// TIA Portal project "pick and place xyz" (V17)
// Vorlageprojekt für das Buch mit Zielsystem S7-1200

(* hardware
DEVICE "S7-1200-Station_1"  S7-1200 Station
   slot 0: "Baugruppenträger_0"  Rack  V1.0
   slot 1: "PLC_1"  CPU 1211C DC/DC/DC  6ES7 211-1AE40-0XB0  V4.1
*)

// ===== PLC "PLC_1"  CPU 1211C DC/DC/DC =====

VAR_GLOBAL   // PLC tag table "Standard-Variablentabelle"
   "box at place" AT %I0.0 : Bool;
   "part at place" AT %I0.1 : Bool;
   "detected" AT %I0.2 : Bool;
   "c limit" AT %I0.3 : Bool;
   "start" AT %I0.4 : Bool;
   "reset" AT %I0.5 : Bool;
   "stop" AT %I0.6 : Bool;
   "e stop" AT %I0.7 : Bool;
   "auto" AT %I1.0 : Bool;
   "FACTORY io run" AT %I1.1 : Bool;
   "x" AT %ID30 : Real;
   "y" AT %ID34 : Real;
   "z" AT %ID38 : Real;
   "box conv" AT %Q0.0 : Bool;
   "part conv" AT %Q0.1 : Bool;
   "exit conv" AT %Q0.2 : Bool;
   "c+" AT %Q0.3 : Bool;
   "grab" AT %Q0.4 : Bool;
   "exit green" AT %Q0.5 : Bool;
   "exit yellow" AT %Q0.6 : Bool;
   "exit red" AT %Q0.7 : Bool;
   "start light" AT %Q1.0 : Bool;
   "reset light" AT %Q1.1 : Bool;
   "stop light" AT %Q1.2 : Bool;
   "sp x" AT %QD30 : Real;
   "sp y" AT %QD34 : Real;
   "sp z" AT %QD38 : Real;
   "count" AT %QD42 : DInt;
   "Tag_1" AT %M0.0 : Bool;
   "Tag_2" AT %M0.1 : Bool;
   "reset count" AT %M0.2 : Bool;
END_VAR

DATA_BLOCK "modes"   // DB2
{ S7_Optimized_Access := 'TRUE' }
VERSION : 0.1
   VAR
      "stop mode" : Bool;
      "start mode" : Bool;
      "auto mode" : Bool;
      "reset mode" : Bool;
      "e stop mode" : Bool;
      "home position" : Bool;
   END_VAR
BEGIN
END_DATA_BLOCK

DATA_BLOCK "steps"   // DB4
{ S7_Optimized_Access := 'TRUE' }
VERSION : 0.1
   VAR
      "next step" : Int := 0;
      "curent step" : Int := 0;
   END_VAR
BEGIN
END_DATA_BLOCK

// folder: System blocks/Program resources

DATA_BLOCK "counter"   // DB1
{ S7_Optimized_Access := 'TRUE' }
AUTHOR : Simatic
FAMILY : IEC
NAME : CNTR
VERSION : 1.0
// stored: InstanceOfName IEC_COUNTER
"IEC_COUNTER"
BEGIN
END_DATA_BLOCK

// folder: (top level)

FUNCTION "1 operation modes" : Void   // FC1, LAD
{ S7_Optimized_Access := 'TRUE' }
VERSION : 0.1
BEGIN

REGION Network 1: start mode
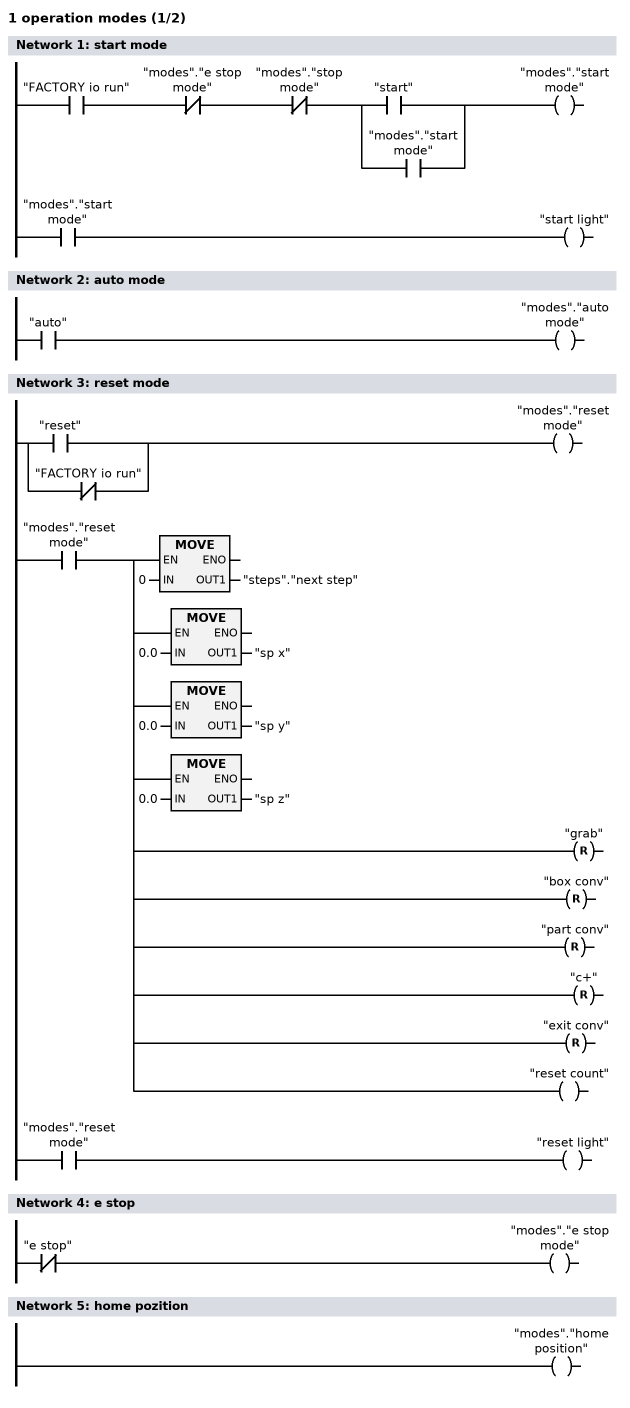
   RUNG wire#powerrail
      Contact( "FACTORY io run" )
      I_Contact( "modes"."e stop mode" )
      I_Contact( "modes"."stop mode" )
      wire#w1
      Contact( "start" )
      wire#w2
      Coil( "modes"."start mode" )
   END_RUNG
   RUNG wire#w1
      Contact( "modes"."start mode" )
   END_RUNG wire#w2
   RUNG wire#powerrail
      Contact( "modes"."start mode" )
      Coil( "start light" )
   END_RUNG
   // the same network as SCL:
   "modes"."start mode" := "FACTORY io run" AND NOT "modes"."e stop mode" AND NOT "modes"."stop mode" AND ("start" OR "modes"."start mode");
   "start light" := "modes"."start mode";
END_REGION

REGION Network 2: auto mode
   RUNG wire#powerrail
      Contact( "auto" )
      Coil( "modes"."auto mode" )
   END_RUNG
   // the same network as SCL:
   "modes"."auto mode" := "auto";
END_REGION

REGION Network 3: reset mode
   RUNG wire#powerrail
      Contact( "reset" )
      wire#w1
      Coil( "modes"."reset mode" )
   END_RUNG
   RUNG wire#powerrail
      I_Contact( "FACTORY io run" )
   END_RUNG wire#w1
   RUNG wire#powerrail
      Contact( "modes"."reset mode" )
      wire#w2
      Move(in := 0, out1 => "steps"."next step")
   END_RUNG
   RUNG wire#w2
      Move(in := 0.0, out1 => "sp x")
   END_RUNG
   RUNG wire#w2
      Move(in := 0.0, out1 => "sp y")
   END_RUNG
   RUNG wire#w2
      Move(in := 0.0, out1 => "sp z")
   END_RUNG
   RUNG wire#w2
      R_Coil( "grab" )
   END_RUNG
   RUNG wire#w2
      R_Coil( "box conv" )
   END_RUNG
   RUNG wire#w2
      R_Coil( "part conv" )
   END_RUNG
   RUNG wire#w2
      R_Coil( "c+" )
   END_RUNG
   RUNG wire#w2
      R_Coil( "exit conv" )
   END_RUNG
   RUNG wire#w2
      Coil( "reset count" )
   END_RUNG
   RUNG wire#powerrail
      Contact( "modes"."reset mode" )
      Coil( "reset light" )
   END_RUNG
   // the same network as SCL:
   "modes"."reset mode" := "reset" OR NOT "FACTORY io run";
   IF "modes"."reset mode" THEN
       "steps"."next step" := 0;
       "sp x" := 0.0;
       "sp y" := 0.0;
       "sp z" := 0.0;
       "grab" := FALSE;
       "box conv" := FALSE;
       "part conv" := FALSE;
       "c+" := FALSE;
       "exit conv" := FALSE;
   END_IF;
   "reset count" := "modes"."reset mode";
   "reset light" := "modes"."reset mode";
END_REGION

REGION Network 4: e stop
   RUNG wire#powerrail
      I_Contact( "e stop" )
      Coil( "modes"."e stop mode" )
   END_RUNG
   // the same network as SCL:
   "modes"."e stop mode" := NOT "e stop";
END_REGION

REGION Network 5: home pozition
   RUNG wire#powerrail
      Coil( "modes"."home position" )
   END_RUNG
   // the same network as SCL:
   "modes"."home position" := TRUE;
END_REGION

REGION Network 6
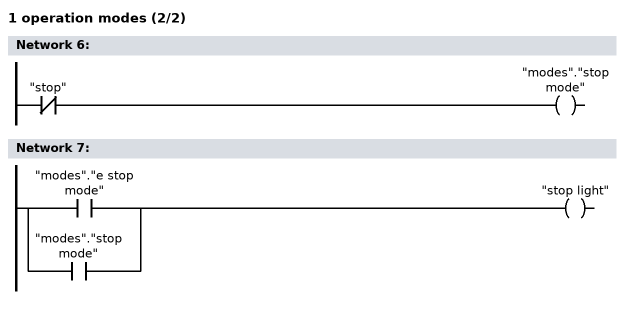
   RUNG wire#powerrail
      I_Contact( "stop" )
      Coil( "modes"."stop mode" )
   END_RUNG
   // the same network as SCL:
   "modes"."stop mode" := NOT "stop";
END_REGION

REGION Network 7
   RUNG wire#powerrail
      Contact( "modes"."e stop mode" )
      wire#w1
      Coil( "stop light" )
   END_RUNG
   RUNG wire#powerrail
      Contact( "modes"."stop mode" )
   END_RUNG wire#w1
   // the same network as SCL:
   "stop light" := "modes"."e stop mode" OR "modes"."stop mode";
END_REGION
END_FUNCTION

FUNCTION "2 step definition" : Void   // FC2, LAD
{ S7_Optimized_Access := 'TRUE' }
VERSION : 0.1
BEGIN

REGION Network 1
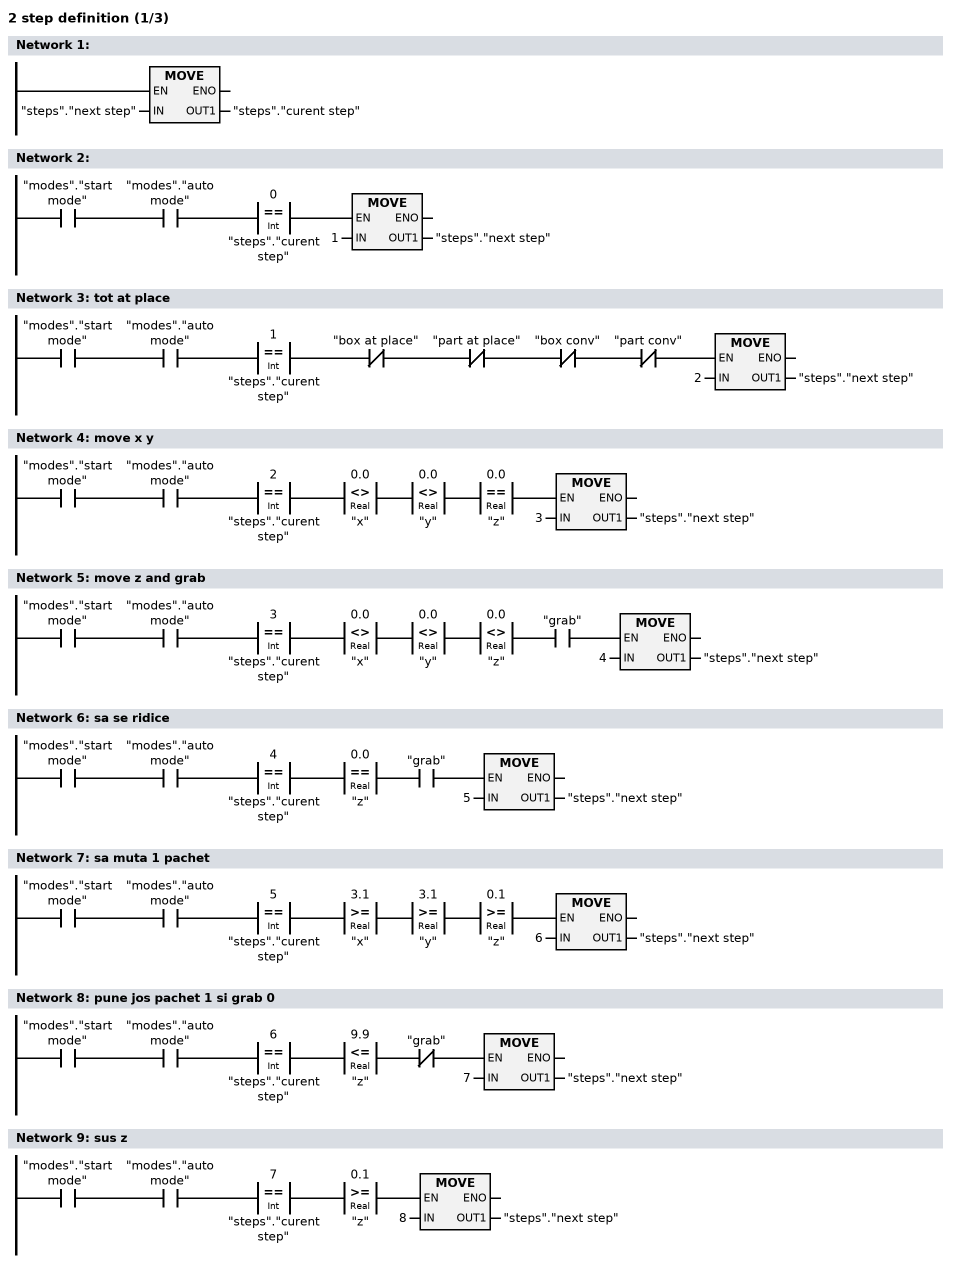
   RUNG wire#powerrail
      Move(in := "steps"."next step", out1 => "steps"."curent step")
   END_RUNG
   // the same network as SCL:
   "steps"."curent step" := "steps"."next step";
END_REGION

REGION Network 2
   RUNG wire#powerrail
      Contact( "modes"."start mode" )
      Contact( "modes"."auto mode" )
      { S7_Templates := "SrcType := Int" } EQ_Contact(in1 := 0, in2 := "steps"."curent step")
      Move(in := 1, out1 => "steps"."next step")
   END_RUNG
   // the same network as SCL:
   IF "modes"."start mode" AND "modes"."auto mode" AND (0 = "steps"."curent step") THEN
       "steps"."next step" := 1;
   END_IF;
END_REGION

REGION Network 3: tot at place
   RUNG wire#powerrail
      Contact( "modes"."start mode" )
      Contact( "modes"."auto mode" )
      { S7_Templates := "SrcType := Int" } EQ_Contact(in1 := 1, in2 := "steps"."curent step")
      I_Contact( "box at place" )
      I_Contact( "part at place" )
      I_Contact( "box conv" )
      I_Contact( "part conv" )
      Move(in := 2, out1 => "steps"."next step")
   END_RUNG
   // the same network as SCL:
   IF "modes"."start mode" AND "modes"."auto mode" AND (1 = "steps"."curent step") AND NOT "box at place" AND NOT "part at place" AND NOT "box conv" AND NOT "part conv" THEN
       "steps"."next step" := 2;
   END_IF;
END_REGION

REGION Network 4: move x y
   RUNG wire#powerrail
      Contact( "modes"."start mode" )
      Contact( "modes"."auto mode" )
      { S7_Templates := "SrcType := Int" } EQ_Contact(in1 := 2, in2 := "steps"."curent step")
      { S7_Templates := "SrcType := Real" } NE_Contact(in1 := 0.0, in2 := "x")
      { S7_Templates := "SrcType := Real" } NE_Contact(in1 := 0.0, in2 := "y")
      { S7_Templates := "SrcType := Real" } EQ_Contact(in1 := 0.0, in2 := "z")
      Move(in := 3, out1 => "steps"."next step")
   END_RUNG
   // the same network as SCL:
   IF "modes"."start mode" AND "modes"."auto mode" AND (2 = "steps"."curent step") AND (0.0 <> "x") AND (0.0 <> "y") AND (0.0 = "z") THEN
       "steps"."next step" := 3;
   END_IF;
END_REGION

REGION Network 5: move z and grab
   RUNG wire#powerrail
      Contact( "modes"."start mode" )
      Contact( "modes"."auto mode" )
      { S7_Templates := "SrcType := Int" } EQ_Contact(in1 := 3, in2 := "steps"."curent step")
      { S7_Templates := "SrcType := Real" } NE_Contact(in1 := 0.0, in2 := "x")
      { S7_Templates := "SrcType := Real" } NE_Contact(in1 := 0.0, in2 := "y")
      { S7_Templates := "SrcType := Real" } NE_Contact(in1 := 0.0, in2 := "z")
      Contact( "grab" )
      Move(in := 4, out1 => "steps"."next step")
   END_RUNG
   // the same network as SCL:
   IF "modes"."start mode" AND "modes"."auto mode" AND (3 = "steps"."curent step") AND (0.0 <> "x") AND (0.0 <> "y") AND (0.0 <> "z") AND "grab" THEN
       "steps"."next step" := 4;
   END_IF;
END_REGION

REGION Network 6: sa se ridice
   RUNG wire#powerrail
      Contact( "modes"."start mode" )
      Contact( "modes"."auto mode" )
      { S7_Templates := "SrcType := Int" } EQ_Contact(in1 := 4, in2 := "steps"."curent step")
      { S7_Templates := "SrcType := Real" } EQ_Contact(in1 := 0.0, in2 := "z")
      Contact( "grab" )
      Move(in := 5, out1 => "steps"."next step")
   END_RUNG
   // the same network as SCL:
   IF "modes"."start mode" AND "modes"."auto mode" AND (4 = "steps"."curent step") AND (0.0 = "z") AND "grab" THEN
       "steps"."next step" := 5;
   END_IF;
END_REGION

REGION Network 7: sa muta 1 pachet
   RUNG wire#powerrail
      Contact( "modes"."start mode" )
      Contact( "modes"."auto mode" )
      { S7_Templates := "SrcType := Int" } EQ_Contact(in1 := 5, in2 := "steps"."curent step")
      { S7_Templates := "SrcType := Real" } GE_Contact(in1 := 3.1, in2 := "x")
      { S7_Templates := "SrcType := Real" } GE_Contact(in1 := 3.1, in2 := "y")
      { S7_Templates := "SrcType := Real" } GE_Contact(in1 := 0.1, in2 := "z")
      Move(in := 6, out1 => "steps"."next step")
   END_RUNG
   // the same network as SCL:
   IF "modes"."start mode" AND "modes"."auto mode" AND (5 = "steps"."curent step") AND (3.1 >= "x") AND (3.1 >= "y") AND (0.1 >= "z") THEN
       "steps"."next step" := 6;
   END_IF;
END_REGION

REGION Network 8: pune jos pachet 1 si grab 0
   RUNG wire#powerrail
      Contact( "modes"."start mode" )
      Contact( "modes"."auto mode" )
      { S7_Templates := "SrcType := Int" } EQ_Contact(in1 := 6, in2 := "steps"."curent step")
      { S7_Templates := "SrcType := Real" } LE_Contact(in1 := 9.9, in2 := "z")
      I_Contact( "grab" )
      Move(in := 7, out1 => "steps"."next step")
   END_RUNG
   // the same network as SCL:
   IF "modes"."start mode" AND "modes"."auto mode" AND (6 = "steps"."curent step") AND (9.9 <= "z") AND NOT "grab" THEN
       "steps"."next step" := 7;
   END_IF;
END_REGION

REGION Network 9: sus z
   RUNG wire#powerrail
      Contact( "modes"."start mode" )
      Contact( "modes"."auto mode" )
      { S7_Templates := "SrcType := Int" } EQ_Contact(in1 := 7, in2 := "steps"."curent step")
      { S7_Templates := "SrcType := Real" } GE_Contact(in1 := 0.1, in2 := "z")
      Move(in := 8, out1 => "steps"."next step")
   END_RUNG
   // the same network as SCL:
   IF "modes"."start mode" AND "modes"."auto mode" AND (7 = "steps"."curent step") AND (0.1 >= "z") THEN
       "steps"."next step" := 8;
   END_IF;
END_REGION

REGION Network 10: xyz at place
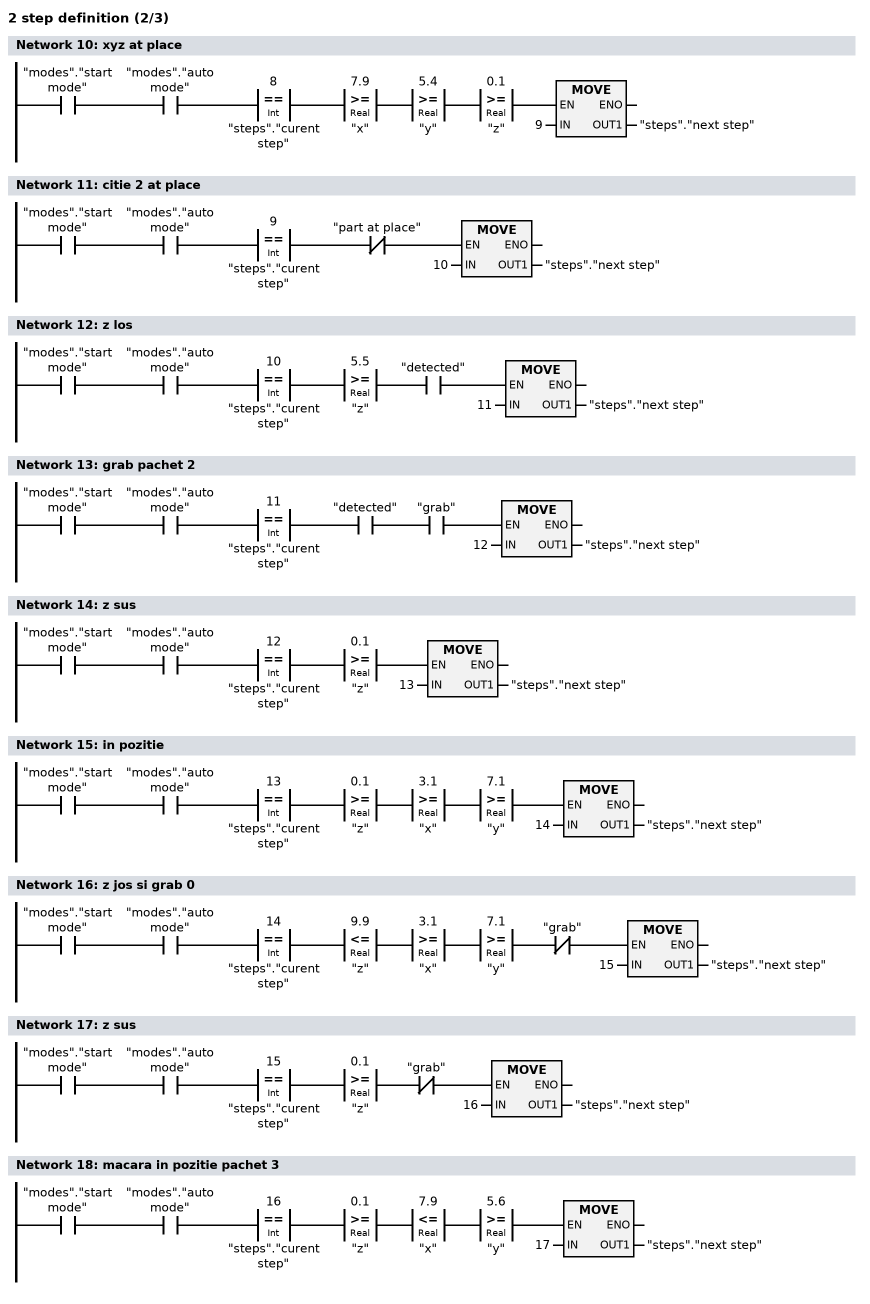
   RUNG wire#powerrail
      Contact( "modes"."start mode" )
      Contact( "modes"."auto mode" )
      { S7_Templates := "SrcType := Int" } EQ_Contact(in1 := 8, in2 := "steps"."curent step")
      { S7_Templates := "SrcType := Real" } GE_Contact(in1 := 7.9, in2 := "x")
      { S7_Templates := "SrcType := Real" } GE_Contact(in1 := 5.4, in2 := "y")
      { S7_Templates := "SrcType := Real" } GE_Contact(in1 := 0.1, in2 := "z")
      Move(in := 9, out1 => "steps"."next step")
   END_RUNG
   // the same network as SCL:
   IF "modes"."start mode" AND "modes"."auto mode" AND (8 = "steps"."curent step") AND (7.9 >= "x") AND (5.4 >= "y") AND (0.1 >= "z") THEN
       "steps"."next step" := 9;
   END_IF;
END_REGION

REGION Network 11: citie 2 at place
   RUNG wire#powerrail
      Contact( "modes"."start mode" )
      Contact( "modes"."auto mode" )
      { S7_Templates := "SrcType := Int" } EQ_Contact(in1 := 9, in2 := "steps"."curent step")
      I_Contact( "part at place" )
      Move(in := 10, out1 => "steps"."next step")
   END_RUNG
   // the same network as SCL:
   IF "modes"."start mode" AND "modes"."auto mode" AND (9 = "steps"."curent step") AND NOT "part at place" THEN
       "steps"."next step" := 10;
   END_IF;
END_REGION

REGION Network 12: z los
   RUNG wire#powerrail
      Contact( "modes"."start mode" )
      Contact( "modes"."auto mode" )
      { S7_Templates := "SrcType := Int" } EQ_Contact(in1 := 10, in2 := "steps"."curent step")
      { S7_Templates := "SrcType := Real" } GE_Contact(in1 := 5.5, in2 := "z")
      Contact( "detected" )
      Move(in := 11, out1 => "steps"."next step")
   END_RUNG
   // the same network as SCL:
   IF "modes"."start mode" AND "modes"."auto mode" AND (10 = "steps"."curent step") AND (5.5 >= "z") AND "detected" THEN
       "steps"."next step" := 11;
   END_IF;
END_REGION

REGION Network 13: grab pachet 2
   RUNG wire#powerrail
      Contact( "modes"."start mode" )
      Contact( "modes"."auto mode" )
      { S7_Templates := "SrcType := Int" } EQ_Contact(in1 := 11, in2 := "steps"."curent step")
      Contact( "detected" )
      Contact( "grab" )
      Move(in := 12, out1 => "steps"."next step")
   END_RUNG
   // the same network as SCL:
   IF "modes"."start mode" AND "modes"."auto mode" AND (11 = "steps"."curent step") AND "detected" AND "grab" THEN
       "steps"."next step" := 12;
   END_IF;
END_REGION

REGION Network 14: z sus
   RUNG wire#powerrail
      Contact( "modes"."start mode" )
      Contact( "modes"."auto mode" )
      { S7_Templates := "SrcType := Int" } EQ_Contact(in1 := 12, in2 := "steps"."curent step")
      { S7_Templates := "SrcType := Real" } GE_Contact(in1 := 0.1, in2 := "z")
      Move(in := 13, out1 => "steps"."next step")
   END_RUNG
   // the same network as SCL:
   IF "modes"."start mode" AND "modes"."auto mode" AND (12 = "steps"."curent step") AND (0.1 >= "z") THEN
       "steps"."next step" := 13;
   END_IF;
END_REGION

REGION Network 15: in pozitie
   RUNG wire#powerrail
      Contact( "modes"."start mode" )
      Contact( "modes"."auto mode" )
      { S7_Templates := "SrcType := Int" } EQ_Contact(in1 := 13, in2 := "steps"."curent step")
      { S7_Templates := "SrcType := Real" } GE_Contact(in1 := 0.1, in2 := "z")
      { S7_Templates := "SrcType := Real" } GE_Contact(in1 := 3.1, in2 := "x")
      { S7_Templates := "SrcType := Real" } GE_Contact(in1 := 7.1, in2 := "y")
      Move(in := 14, out1 => "steps"."next step")
   END_RUNG
   // the same network as SCL:
   IF "modes"."start mode" AND "modes"."auto mode" AND (13 = "steps"."curent step") AND (0.1 >= "z") AND (3.1 >= "x") AND (7.1 >= "y") THEN
       "steps"."next step" := 14;
   END_IF;
END_REGION

REGION Network 16: z jos si grab 0
   RUNG wire#powerrail
      Contact( "modes"."start mode" )
      Contact( "modes"."auto mode" )
      { S7_Templates := "SrcType := Int" } EQ_Contact(in1 := 14, in2 := "steps"."curent step")
      { S7_Templates := "SrcType := Real" } LE_Contact(in1 := 9.9, in2 := "z")
      { S7_Templates := "SrcType := Real" } GE_Contact(in1 := 3.1, in2 := "x")
      { S7_Templates := "SrcType := Real" } GE_Contact(in1 := 7.1, in2 := "y")
      I_Contact( "grab" )
      Move(in := 15, out1 => "steps"."next step")
   END_RUNG
   // the same network as SCL:
   IF "modes"."start mode" AND "modes"."auto mode" AND (14 = "steps"."curent step") AND (9.9 <= "z") AND (3.1 >= "x") AND (7.1 >= "y") AND NOT "grab" THEN
       "steps"."next step" := 15;
   END_IF;
END_REGION

REGION Network 17: z sus
   RUNG wire#powerrail
      Contact( "modes"."start mode" )
      Contact( "modes"."auto mode" )
      { S7_Templates := "SrcType := Int" } EQ_Contact(in1 := 15, in2 := "steps"."curent step")
      { S7_Templates := "SrcType := Real" } GE_Contact(in1 := 0.1, in2 := "z")
      I_Contact( "grab" )
      Move(in := 16, out1 => "steps"."next step")
   END_RUNG
   // the same network as SCL:
   IF "modes"."start mode" AND "modes"."auto mode" AND (15 = "steps"."curent step") AND (0.1 >= "z") AND NOT "grab" THEN
       "steps"."next step" := 16;
   END_IF;
END_REGION

REGION Network 18: macara in pozitie pachet 3
   RUNG wire#powerrail
      Contact( "modes"."start mode" )
      Contact( "modes"."auto mode" )
      { S7_Templates := "SrcType := Int" } EQ_Contact(in1 := 16, in2 := "steps"."curent step")
      { S7_Templates := "SrcType := Real" } GE_Contact(in1 := 0.1, in2 := "z")
      { S7_Templates := "SrcType := Real" } LE_Contact(in1 := 7.9, in2 := "x")
      { S7_Templates := "SrcType := Real" } GE_Contact(in1 := 5.6, in2 := "y")
      Move(in := 17, out1 => "steps"."next step")
   END_RUNG
   // the same network as SCL:
   IF "modes"."start mode" AND "modes"."auto mode" AND (16 = "steps"."curent step") AND (0.1 >= "z") AND (7.9 <= "x") AND (5.6 >= "y") THEN
       "steps"."next step" := 17;
   END_IF;
END_REGION

REGION Network 19: part 3 in pozitie
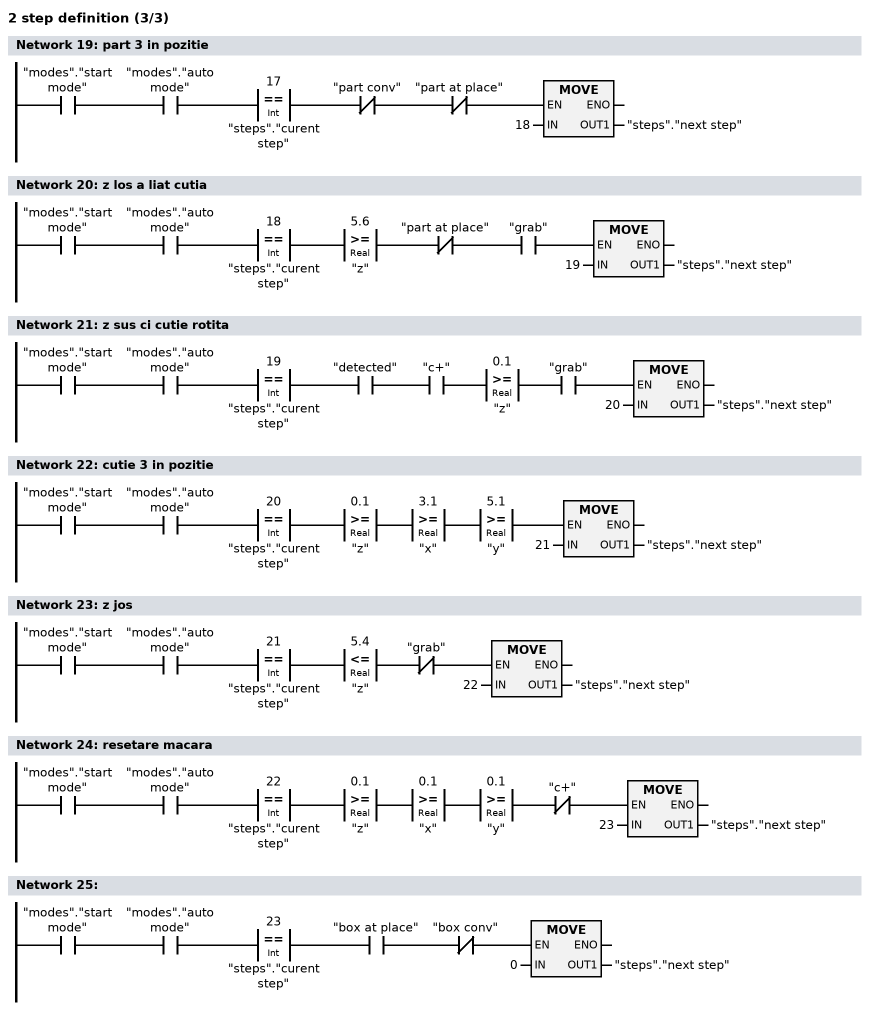
   RUNG wire#powerrail
      Contact( "modes"."start mode" )
      Contact( "modes"."auto mode" )
      { S7_Templates := "SrcType := Int" } EQ_Contact(in1 := 17, in2 := "steps"."curent step")
      I_Contact( "part conv" )
      I_Contact( "part at place" )
      Move(in := 18, out1 => "steps"."next step")
   END_RUNG
   // the same network as SCL:
   IF "modes"."start mode" AND "modes"."auto mode" AND (17 = "steps"."curent step") AND NOT "part conv" AND NOT "part at place" THEN
       "steps"."next step" := 18;
   END_IF;
END_REGION

REGION Network 20: z los a liat cutia
   RUNG wire#powerrail
      Contact( "modes"."start mode" )
      Contact( "modes"."auto mode" )
      { S7_Templates := "SrcType := Int" } EQ_Contact(in1 := 18, in2 := "steps"."curent step")
      { S7_Templates := "SrcType := Real" } GE_Contact(in1 := 5.6, in2 := "z")
      I_Contact( "part at place" )
      Contact( "grab" )
      Move(in := 19, out1 => "steps"."next step")
   END_RUNG
   // the same network as SCL:
   IF "modes"."start mode" AND "modes"."auto mode" AND (18 = "steps"."curent step") AND (5.6 >= "z") AND NOT "part at place" AND "grab" THEN
       "steps"."next step" := 19;
   END_IF;
END_REGION

REGION Network 21: z sus ci cutie rotita
   RUNG wire#powerrail
      Contact( "modes"."start mode" )
      Contact( "modes"."auto mode" )
      { S7_Templates := "SrcType := Int" } EQ_Contact(in1 := 19, in2 := "steps"."curent step")
      Contact( "detected" )
      Contact( "c+" )
      { S7_Templates := "SrcType := Real" } GE_Contact(in1 := 0.1, in2 := "z")
      Contact( "grab" )
      Move(in := 20, out1 => "steps"."next step")
   END_RUNG
   // the same network as SCL:
   IF "modes"."start mode" AND "modes"."auto mode" AND (19 = "steps"."curent step") AND "detected" AND "c+" AND (0.1 >= "z") AND "grab" THEN
       "steps"."next step" := 20;
   END_IF;
END_REGION

REGION Network 22: cutie 3 in pozitie
   RUNG wire#powerrail
      Contact( "modes"."start mode" )
      Contact( "modes"."auto mode" )
      { S7_Templates := "SrcType := Int" } EQ_Contact(in1 := 20, in2 := "steps"."curent step")
      { S7_Templates := "SrcType := Real" } GE_Contact(in1 := 0.1, in2 := "z")
      { S7_Templates := "SrcType := Real" } GE_Contact(in1 := 3.1, in2 := "x")
      { S7_Templates := "SrcType := Real" } GE_Contact(in1 := 5.1, in2 := "y")
      Move(in := 21, out1 => "steps"."next step")
   END_RUNG
   // the same network as SCL:
   IF "modes"."start mode" AND "modes"."auto mode" AND (20 = "steps"."curent step") AND (0.1 >= "z") AND (3.1 >= "x") AND (5.1 >= "y") THEN
       "steps"."next step" := 21;
   END_IF;
END_REGION

REGION Network 23: z jos
   RUNG wire#powerrail
      Contact( "modes"."start mode" )
      Contact( "modes"."auto mode" )
      { S7_Templates := "SrcType := Int" } EQ_Contact(in1 := 21, in2 := "steps"."curent step")
      { S7_Templates := "SrcType := Real" } LE_Contact(in1 := 5.4, in2 := "z")
      I_Contact( "grab" )
      Move(in := 22, out1 => "steps"."next step")
   END_RUNG
   // the same network as SCL:
   IF "modes"."start mode" AND "modes"."auto mode" AND (21 = "steps"."curent step") AND (5.4 <= "z") AND NOT "grab" THEN
       "steps"."next step" := 22;
   END_IF;
END_REGION

REGION Network 24: resetare macara
   RUNG wire#powerrail
      Contact( "modes"."start mode" )
      Contact( "modes"."auto mode" )
      { S7_Templates := "SrcType := Int" } EQ_Contact(in1 := 22, in2 := "steps"."curent step")
      { S7_Templates := "SrcType := Real" } GE_Contact(in1 := 0.1, in2 := "z")
      { S7_Templates := "SrcType := Real" } GE_Contact(in1 := 0.1, in2 := "x")
      { S7_Templates := "SrcType := Real" } GE_Contact(in1 := 0.1, in2 := "y")
      I_Contact( "c+" )
      Move(in := 23, out1 => "steps"."next step")
   END_RUNG
   // the same network as SCL:
   IF "modes"."start mode" AND "modes"."auto mode" AND (22 = "steps"."curent step") AND (0.1 >= "z") AND (0.1 >= "x") AND (0.1 >= "y") AND NOT "c+" THEN
       "steps"."next step" := 23;
   END_IF;
END_REGION

REGION Network 25
   RUNG wire#powerrail
      Contact( "modes"."start mode" )
      Contact( "modes"."auto mode" )
      { S7_Templates := "SrcType := Int" } EQ_Contact(in1 := 23, in2 := "steps"."curent step")
      Contact( "box at place" )
      I_Contact( "box conv" )
      Move(in := 0, out1 => "steps"."next step")
   END_RUNG
   // the same network as SCL:
   IF "modes"."start mode" AND "modes"."auto mode" AND (23 = "steps"."curent step") AND "box at place" AND NOT "box conv" THEN
       "steps"."next step" := 0;
   END_IF;
END_REGION
END_FUNCTION

FUNCTION "3 step execution" : Void   // FC3, LAD
{ S7_Optimized_Access := 'TRUE' }
VERSION : 0.1
   VAR_TEMP   // added for the SCL form of the ladder/FBD networks
      _w1 : Bool;
   END_VAR
BEGIN

REGION Network 1
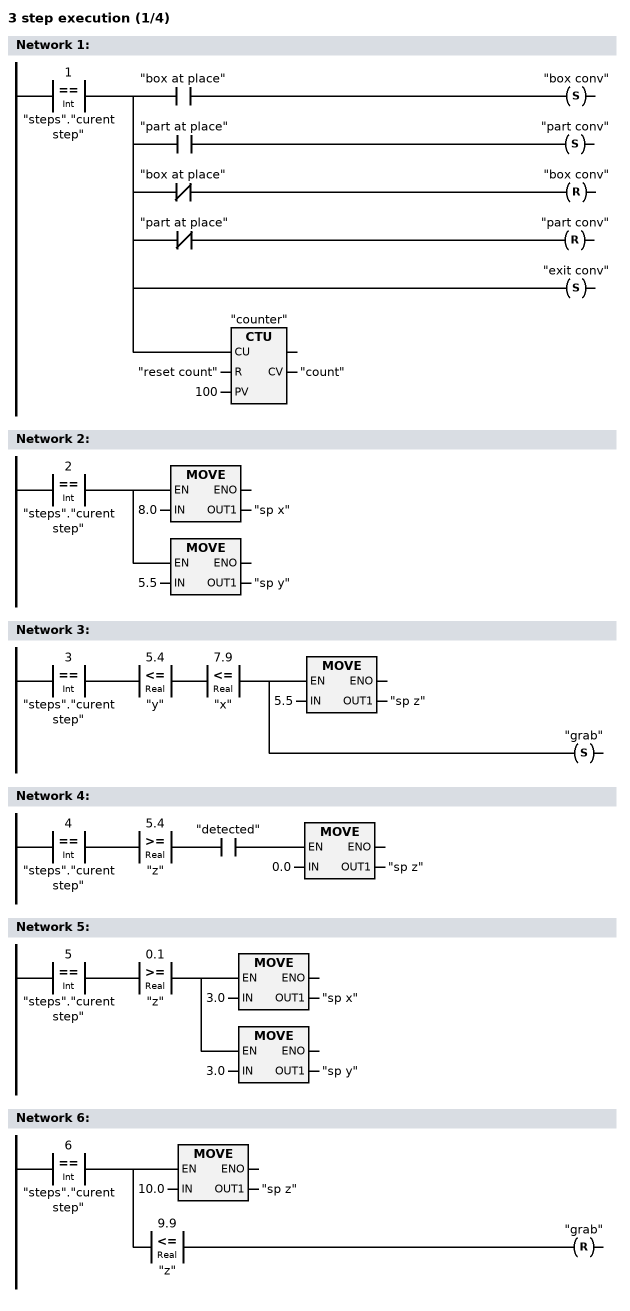
   #_w1 := 1 = "steps"."curent step";
   IF #_w1 AND "box at place" THEN "box conv" := TRUE; END_IF;
   IF #_w1 AND "part at place" THEN "part conv" := TRUE; END_IF;
   IF #_w1 AND NOT "box at place" THEN "box conv" := FALSE; END_IF;
   IF #_w1 AND NOT "part at place" THEN "part conv" := FALSE; END_IF;
   IF #_w1 THEN "exit conv" := TRUE; END_IF;
   "counter".CTU(CU := #_w1, R := "reset count", PV := 100, CV => "count");
END_REGION

REGION Network 2
   RUNG wire#powerrail
      { S7_Templates := "SrcType := Int" } EQ_Contact(in1 := 2, in2 := "steps"."curent step")
      wire#w1
      Move(in := 8.0, out1 => "sp x")
   END_RUNG
   RUNG wire#w1
      Move(in := 5.5, out1 => "sp y")
   END_RUNG
   // the same network as SCL:
   IF 2 = "steps"."curent step" THEN
       "sp x" := 8.0;
       "sp y" := 5.5;
   END_IF;
END_REGION

REGION Network 3
   RUNG wire#powerrail
      { S7_Templates := "SrcType := Int" } EQ_Contact(in1 := 3, in2 := "steps"."curent step")
      { S7_Templates := "SrcType := Real" } LE_Contact(in1 := 5.4, in2 := "y")
      { S7_Templates := "SrcType := Real" } LE_Contact(in1 := 7.9, in2 := "x")
      wire#w1
      Move(in := 5.5, out1 => "sp z")
   END_RUNG
   RUNG wire#w1
      S_Coil( "grab" )
   END_RUNG
   // the same network as SCL:
   IF (3 = "steps"."curent step") AND (5.4 <= "y") AND (7.9 <= "x") THEN
       "sp z" := 5.5;
       "grab" := TRUE;
   END_IF;
END_REGION

REGION Network 4
   RUNG wire#powerrail
      { S7_Templates := "SrcType := Int" } EQ_Contact(in1 := 4, in2 := "steps"."curent step")
      { S7_Templates := "SrcType := Real" } GE_Contact(in1 := 5.4, in2 := "z")
      Contact( "detected" )
      Move(in := 0.0, out1 => "sp z")
   END_RUNG
   // the same network as SCL:
   IF (4 = "steps"."curent step") AND (5.4 >= "z") AND "detected" THEN "sp z" := 0.0; END_IF;
END_REGION

REGION Network 5
   RUNG wire#powerrail
      { S7_Templates := "SrcType := Int" } EQ_Contact(in1 := 5, in2 := "steps"."curent step")
      { S7_Templates := "SrcType := Real" } GE_Contact(in1 := 0.1, in2 := "z")
      wire#w1
      Move(in := 3.0, out1 => "sp x")
   END_RUNG
   RUNG wire#w1
      Move(in := 3.0, out1 => "sp y")
   END_RUNG
   // the same network as SCL:
   IF (5 = "steps"."curent step") AND (0.1 >= "z") THEN
       "sp x" := 3.0;
       "sp y" := 3.0;
   END_IF;
END_REGION

REGION Network 6
   RUNG wire#powerrail
      { S7_Templates := "SrcType := Int" } EQ_Contact(in1 := 6, in2 := "steps"."curent step")
      wire#w1
      Move(in := 10.0, out1 => "sp z")
   END_RUNG
   RUNG wire#w1
      { S7_Templates := "SrcType := Real" } LE_Contact(in1 := 9.9, in2 := "z")
      R_Coil( "grab" )
   END_RUNG
   // the same network as SCL:
   #_w1 := 6 = "steps"."curent step";
   IF #_w1 THEN "sp z" := 10.0; END_IF;
   IF #_w1 AND (9.9 <= "z") THEN "grab" := FALSE; END_IF;
END_REGION

REGION Network 7
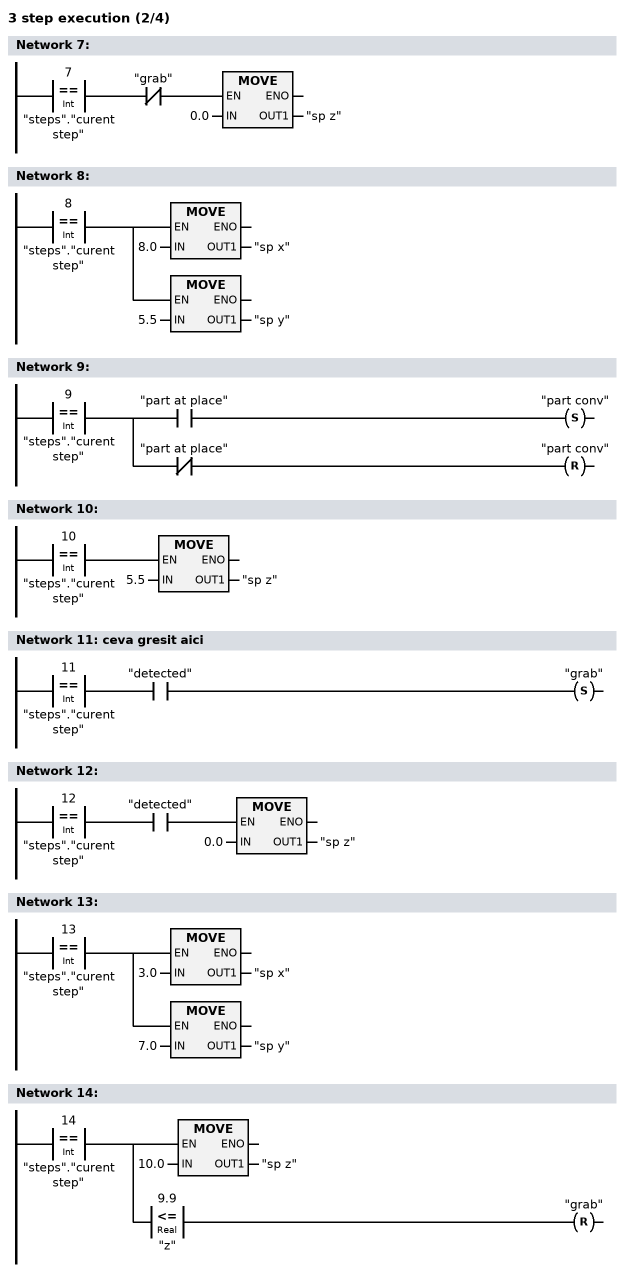
   RUNG wire#powerrail
      { S7_Templates := "SrcType := Int" } EQ_Contact(in1 := 7, in2 := "steps"."curent step")
      I_Contact( "grab" )
      Move(in := 0.0, out1 => "sp z")
   END_RUNG
   // the same network as SCL:
   IF (7 = "steps"."curent step") AND NOT "grab" THEN "sp z" := 0.0; END_IF;
END_REGION

REGION Network 8
   RUNG wire#powerrail
      { S7_Templates := "SrcType := Int" } EQ_Contact(in1 := 8, in2 := "steps"."curent step")
      wire#w1
      Move(in := 8.0, out1 => "sp x")
   END_RUNG
   RUNG wire#w1
      Move(in := 5.5, out1 => "sp y")
   END_RUNG
   // the same network as SCL:
   IF 8 = "steps"."curent step" THEN
       "sp x" := 8.0;
       "sp y" := 5.5;
   END_IF;
END_REGION

REGION Network 9
   RUNG wire#powerrail
      { S7_Templates := "SrcType := Int" } EQ_Contact(in1 := 9, in2 := "steps"."curent step")
      wire#w1
      Contact( "part at place" )
      S_Coil( "part conv" )
   END_RUNG
   RUNG wire#w1
      I_Contact( "part at place" )
      R_Coil( "part conv" )
   END_RUNG
   // the same network as SCL:
   #_w1 := 9 = "steps"."curent step";
   IF #_w1 AND "part at place" THEN "part conv" := TRUE; END_IF;
   IF #_w1 AND NOT "part at place" THEN "part conv" := FALSE; END_IF;
END_REGION

REGION Network 10
   RUNG wire#powerrail
      { S7_Templates := "SrcType := Int" } EQ_Contact(in1 := 10, in2 := "steps"."curent step")
      Move(in := 5.5, out1 => "sp z")
   END_RUNG
   // the same network as SCL:
   IF 10 = "steps"."curent step" THEN "sp z" := 5.5; END_IF;
END_REGION

REGION Network 11: ceva gresit aici
   RUNG wire#powerrail
      { S7_Templates := "SrcType := Int" } EQ_Contact(in1 := 11, in2 := "steps"."curent step")
      Contact( "detected" )
      S_Coil( "grab" )
   END_RUNG
   // the same network as SCL:
   IF (11 = "steps"."curent step") AND "detected" THEN "grab" := TRUE; END_IF;
END_REGION

REGION Network 12
   RUNG wire#powerrail
      { S7_Templates := "SrcType := Int" } EQ_Contact(in1 := 12, in2 := "steps"."curent step")
      Contact( "detected" )
      Move(in := 0.0, out1 => "sp z")
   END_RUNG
   // the same network as SCL:
   IF (12 = "steps"."curent step") AND "detected" THEN "sp z" := 0.0; END_IF;
END_REGION

REGION Network 13
   RUNG wire#powerrail
      { S7_Templates := "SrcType := Int" } EQ_Contact(in1 := 13, in2 := "steps"."curent step")
      wire#w1
      Move(in := 3.0, out1 => "sp x")
   END_RUNG
   RUNG wire#w1
      Move(in := 7.0, out1 => "sp y")
   END_RUNG
   // the same network as SCL:
   IF 13 = "steps"."curent step" THEN
       "sp x" := 3.0;
       "sp y" := 7.0;
   END_IF;
END_REGION

REGION Network 14
   RUNG wire#powerrail
      { S7_Templates := "SrcType := Int" } EQ_Contact(in1 := 14, in2 := "steps"."curent step")
      wire#w1
      Move(in := 10.0, out1 => "sp z")
   END_RUNG
   RUNG wire#w1
      { S7_Templates := "SrcType := Real" } LE_Contact(in1 := 9.9, in2 := "z")
      R_Coil( "grab" )
   END_RUNG
   // the same network as SCL:
   #_w1 := 14 = "steps"."curent step";
   IF #_w1 THEN "sp z" := 10.0; END_IF;
   IF #_w1 AND (9.9 <= "z") THEN "grab" := FALSE; END_IF;
END_REGION

REGION Network 15
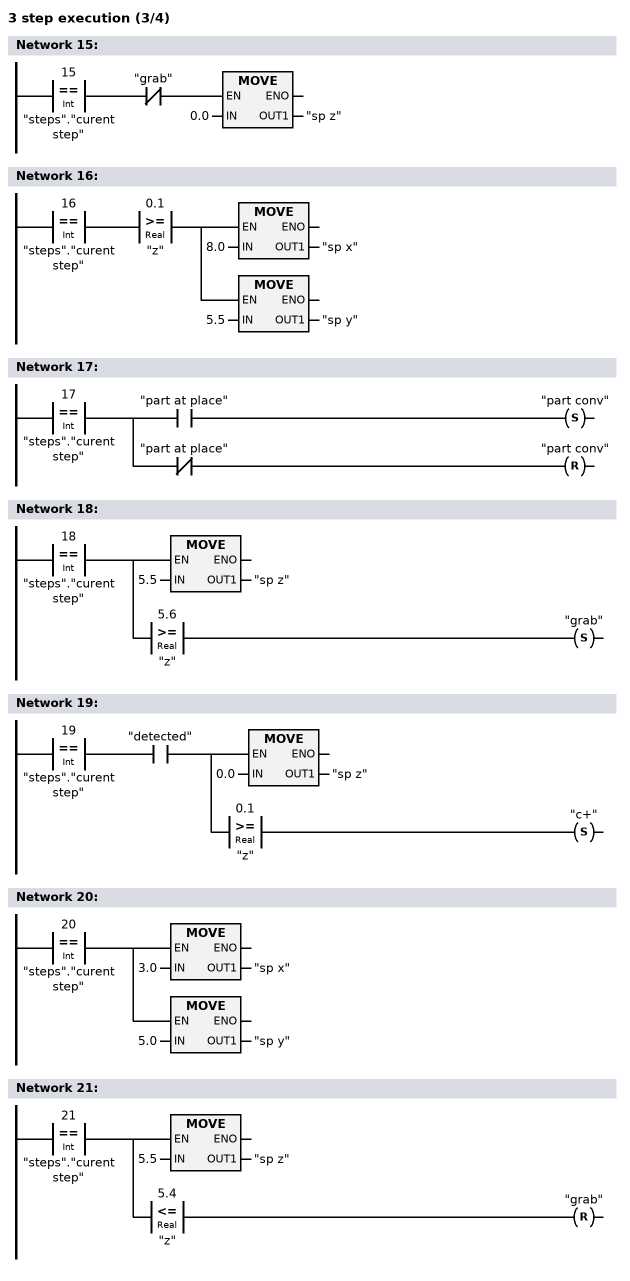
   RUNG wire#powerrail
      { S7_Templates := "SrcType := Int" } EQ_Contact(in1 := 15, in2 := "steps"."curent step")
      I_Contact( "grab" )
      Move(in := 0.0, out1 => "sp z")
   END_RUNG
   // the same network as SCL:
   IF (15 = "steps"."curent step") AND NOT "grab" THEN "sp z" := 0.0; END_IF;
END_REGION

REGION Network 16
   RUNG wire#powerrail
      { S7_Templates := "SrcType := Int" } EQ_Contact(in1 := 16, in2 := "steps"."curent step")
      { S7_Templates := "SrcType := Real" } GE_Contact(in1 := 0.1, in2 := "z")
      wire#w1
      Move(in := 8.0, out1 => "sp x")
   END_RUNG
   RUNG wire#w1
      Move(in := 5.5, out1 => "sp y")
   END_RUNG
   // the same network as SCL:
   IF (16 = "steps"."curent step") AND (0.1 >= "z") THEN
       "sp x" := 8.0;
       "sp y" := 5.5;
   END_IF;
END_REGION

REGION Network 17
   RUNG wire#powerrail
      { S7_Templates := "SrcType := Int" } EQ_Contact(in1 := 17, in2 := "steps"."curent step")
      wire#w1
      Contact( "part at place" )
      S_Coil( "part conv" )
   END_RUNG
   RUNG wire#w1
      I_Contact( "part at place" )
      R_Coil( "part conv" )
   END_RUNG
   // the same network as SCL:
   #_w1 := 17 = "steps"."curent step";
   IF #_w1 AND "part at place" THEN "part conv" := TRUE; END_IF;
   IF #_w1 AND NOT "part at place" THEN "part conv" := FALSE; END_IF;
END_REGION

REGION Network 18
   RUNG wire#powerrail
      { S7_Templates := "SrcType := Int" } EQ_Contact(in1 := 18, in2 := "steps"."curent step")
      wire#w1
      Move(in := 5.5, out1 => "sp z")
   END_RUNG
   RUNG wire#w1
      { S7_Templates := "SrcType := Real" } GE_Contact(in1 := 5.6, in2 := "z")
      S_Coil( "grab" )
   END_RUNG
   // the same network as SCL:
   #_w1 := 18 = "steps"."curent step";
   IF #_w1 THEN "sp z" := 5.5; END_IF;
   IF #_w1 AND (5.6 >= "z") THEN "grab" := TRUE; END_IF;
END_REGION

REGION Network 19
   RUNG wire#powerrail
      { S7_Templates := "SrcType := Int" } EQ_Contact(in1 := 19, in2 := "steps"."curent step")
      Contact( "detected" )
      wire#w1
      Move(in := 0.0, out1 => "sp z")
   END_RUNG
   RUNG wire#w1
      { S7_Templates := "SrcType := Real" } GE_Contact(in1 := 0.1, in2 := "z")
      S_Coil( "c+" )
   END_RUNG
   // the same network as SCL:
   #_w1 := (19 = "steps"."curent step") AND "detected";
   IF #_w1 THEN "sp z" := 0.0; END_IF;
   IF #_w1 AND (0.1 >= "z") THEN "c+" := TRUE; END_IF;
END_REGION

REGION Network 20
   RUNG wire#powerrail
      { S7_Templates := "SrcType := Int" } EQ_Contact(in1 := 20, in2 := "steps"."curent step")
      wire#w1
      Move(in := 3.0, out1 => "sp x")
   END_RUNG
   RUNG wire#w1
      Move(in := 5.0, out1 => "sp y")
   END_RUNG
   // the same network as SCL:
   IF 20 = "steps"."curent step" THEN
       "sp x" := 3.0;
       "sp y" := 5.0;
   END_IF;
END_REGION

REGION Network 21
   RUNG wire#powerrail
      { S7_Templates := "SrcType := Int" } EQ_Contact(in1 := 21, in2 := "steps"."curent step")
      wire#w1
      Move(in := 5.5, out1 => "sp z")
   END_RUNG
   RUNG wire#w1
      { S7_Templates := "SrcType := Real" } LE_Contact(in1 := 5.4, in2 := "z")
      R_Coil( "grab" )
   END_RUNG
   // the same network as SCL:
   #_w1 := 21 = "steps"."curent step";
   IF #_w1 THEN "sp z" := 5.5; END_IF;
   IF #_w1 AND (5.4 <= "z") THEN "grab" := FALSE; END_IF;
END_REGION

REGION Network 22
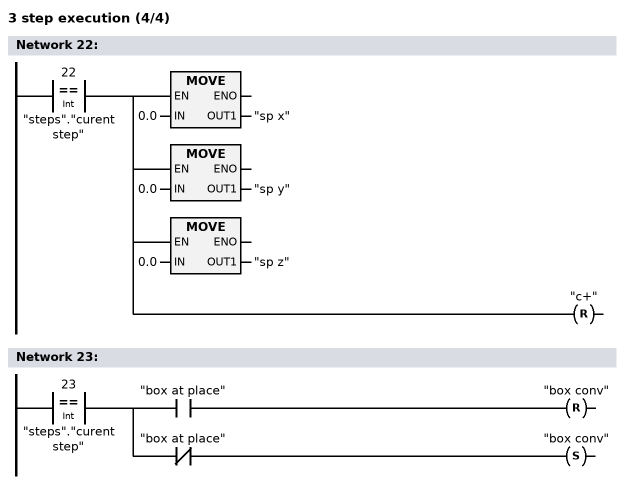
   RUNG wire#powerrail
      { S7_Templates := "SrcType := Int" } EQ_Contact(in1 := 22, in2 := "steps"."curent step")
      wire#w1
      Move(in := 0.0, out1 => "sp x")
   END_RUNG
   RUNG wire#w1
      Move(in := 0.0, out1 => "sp y")
   END_RUNG
   RUNG wire#w1
      Move(in := 0.0, out1 => "sp z")
   END_RUNG
   RUNG wire#w1
      R_Coil( "c+" )
   END_RUNG
   // the same network as SCL:
   IF 22 = "steps"."curent step" THEN
       "sp x" := 0.0;
       "sp y" := 0.0;
       "sp z" := 0.0;
       "c+" := FALSE;
   END_IF;
END_REGION

REGION Network 23
   RUNG wire#powerrail
      { S7_Templates := "SrcType := Int" } EQ_Contact(in1 := 23, in2 := "steps"."curent step")
      wire#w1
      Contact( "box at place" )
      R_Coil( "box conv" )
   END_RUNG
   RUNG wire#w1
      I_Contact( "box at place" )
      S_Coil( "box conv" )
   END_RUNG
   // the same network as SCL:
   #_w1 := 23 = "steps"."curent step";
   IF #_w1 AND "box at place" THEN "box conv" := FALSE; END_IF;
   IF #_w1 AND NOT "box at place" THEN "box conv" := TRUE; END_IF;
END_REGION
END_FUNCTION

FUNCTION "4 output assigment" : Void   // FC4, LAD
{ S7_Optimized_Access := 'TRUE' }
VERSION : 0.1
BEGIN
END_FUNCTION

FUNCTION "MHJ-PLC-Lab-Function-S71200" : Void   // FC9000, SCL
{ S7_Optimized_Access := 'TRUE' }
VERSION : 0.1
   VAR_TEMP
      rdTimeReturn : Int;
      outputTime : DTL;
      SyncVal : Byte;
      forVal : Int;
      forVal_2 : Int;
      Value : Byte;
   END_VAR
   VAR CONSTANT
      CompVal : Byte := 16#34;
      Value_01 : Byte := 16#11;
      Value_01_DW : DWord := 16#A165_D992;
      Value_02_DW : DWord := 16#58BE_4401;
   END_VAR
BEGIN

   #Value:=PEEK(area := 16#82,
        dbNumber := 0,
        byteOffset := 511);
   #Value := #Value + 1;

   POKE(area := 16#82,
        dbNumber := 0,
        byteOffset := 511,
        value := #Value);

   POKE(area:=16#81,
        dbNumber:=0,
        byteOffset:=1016,
        value:=#Value_01_DW);
   POKE(area := 16#81,
        dbNumber := 0,
        byteOffset := 1020,
        value := #Value_02_DW);

   POKE(area := 16#81,
        dbNumber := 0,
        byteOffset := 511,
        value := B#16#00);

   FOR #forVal := 0 TO 120 DO
       FOR #forVal_2:=0 TO 10 DO
           #rdTimeReturn:=RD_SYS_T(#outputTime);
           #rdTimeReturn := WR_SYS_T(#outputTime);
           #rdTimeReturn := RD_SYS_T(#outputTime);
           #rdTimeReturn := WR_SYS_T(#outputTime);
       END_FOR;
       #SyncVal:= PEEK(area := 16#81,
                      dbNumber := 0,
                      byteOffset := 511);
       IF #SyncVal = #CompVal THEN
          GOTO M_1;
       END_IF;
   END_FOR;
   RETURN;

   M_1:
   POKE(area := 16#81,
        dbNumber := 0,
        byteOffset := 511,
        value := B#16#0);
END_FUNCTION

ORGANIZATION_BLOCK "Main"   // OB1, FBD, ProgramCycle
TITLE = "Main Program Sweep (Cycle)"
{ S7_Optimized_Access := 'TRUE' }
VERSION : 0.1
   VAR_INPUT
      Initial_Call : Bool;   // Initial call of this OB
      Remanence : Bool;   // =True, if remanent data are available
   END_VAR
BEGIN

REGION Network 1: Konnektierungsbaustein für PLC-Lab
   // Im Netzwerk 1 wird der Konnektierungsbaustein für PLC-Lab aufgerufen.
   // Dieser Aufruf darf nicht entfernt werden!
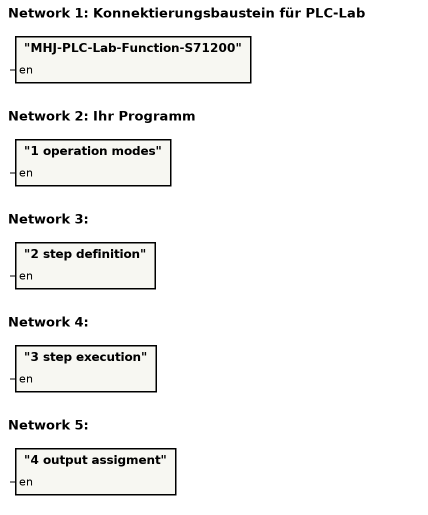
   "MHJ-PLC-Lab-Function-S71200"();
END_REGION

REGION Network 2: Ihr Programm
   // Schreiben Sie ab Netzwerk 2 Ihr Programm
   "1 operation modes"();
END_REGION

REGION Network 3
   "2 step definition"();
END_REGION

REGION Network 4
   "3 step execution"();
END_REGION

REGION Network 5
   "4 output assigment"();
END_REGION
END_ORGANIZATION_BLOCK